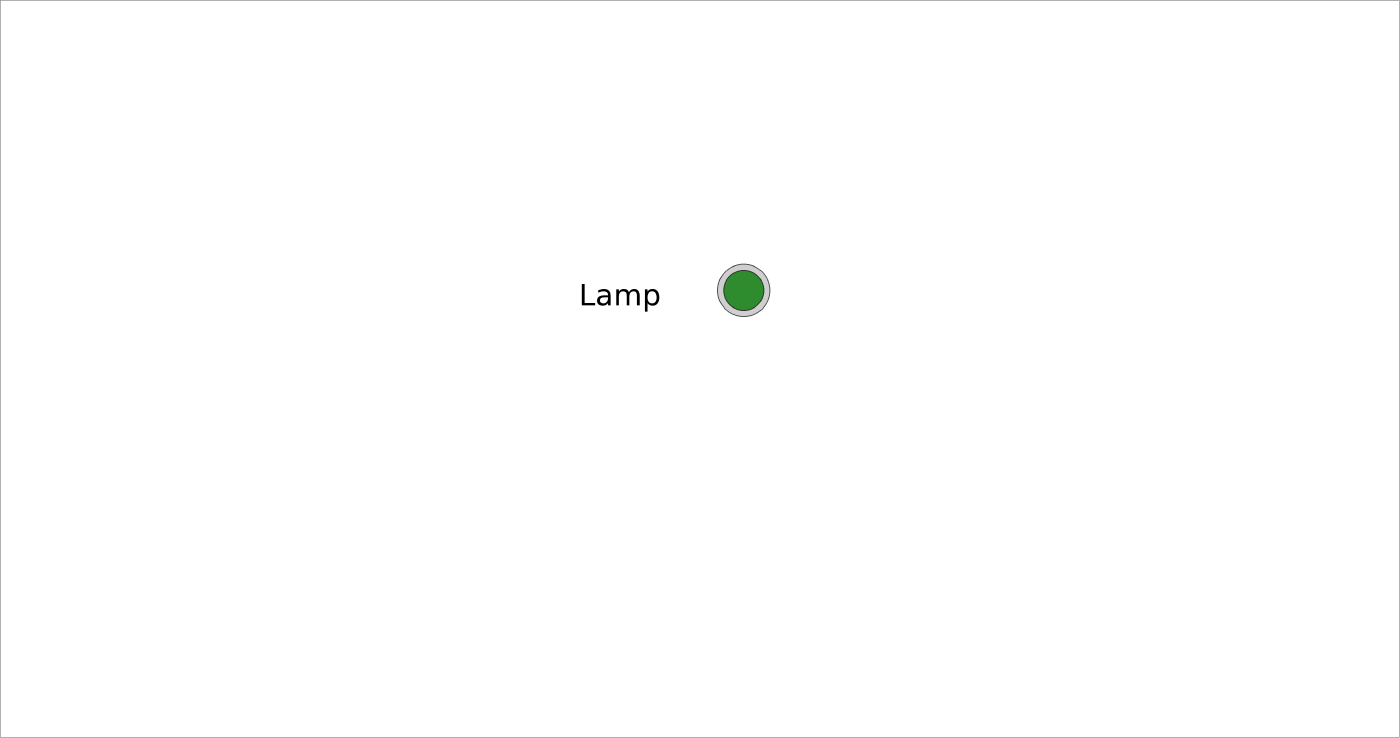
VISUALIZATION visu_sample  // 2048x1080
    Lamp1 (1043,380 90x90), variable: GVL.fb_sample.lamp, style: Lamp-Lamp1-Green
    Label (850,387 120x90), "Lamp"
END_VISUALIZATION

(* stored: Version 1.1.0.1, ProductVersion 3.1.4024.12
   Visu visu_sample: Id {4a2c74dd-6e4c-4dbf-b80f-55c88e9652a0} *)
